(* Schneider Machine Expert - Basic project 06b_counter, file version 3.0.0.0 *)
(* ProjectInformations: Name=New project *)

HARDWARE
  Cpu 0: TM221C40U
  EthernetConfiguration: NetworkName=M221, IpAllocationMode=FixedAddress, IpAddress=0.0.0.0, SubnetMask=0.0.0.0
  SerialLineConfiguration: Baud=Baud19200, Parity=ParityEven, DataBits=DataBits8, StopBits=StopBits1, PhysicalMedium=PhysicalMediumRs485, TransmissionMode=TransmissionModeModbusRtu, SlaveId=1, Addressing=SlaveAddressing
  MastTask: UsePeriodScanMode=false, PeriodScan=100
  FastTask: Period=255
  CpuBehavior: StartingMode=StartAsPreviousState, AutoSaveRamOnEeprom=true, WatchdogPeriod=250

SYMBOLS  (address, symbol, comment, settings)
  %C0         [Preset=10]

POU New POU
  (* SectionNumber=0 *)

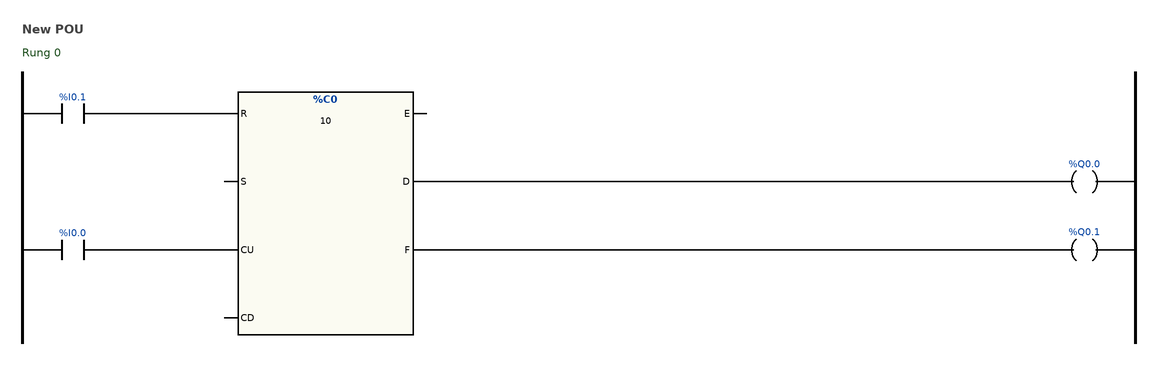

// Rung 0
  BLK %C0
  LD %I0.1
  R
  LD %I0.0
  CU
  OUT_BLK
  LD D
  ST %Q0.0
  LD F
  ST %Q0.1
  END_BLK
  // as ST:
  //   %C0(R := %I0.1, CU := %I0.0);
  //   %Q0.0 := %C0.D;
  //   %Q0.1 := %C0.F;
